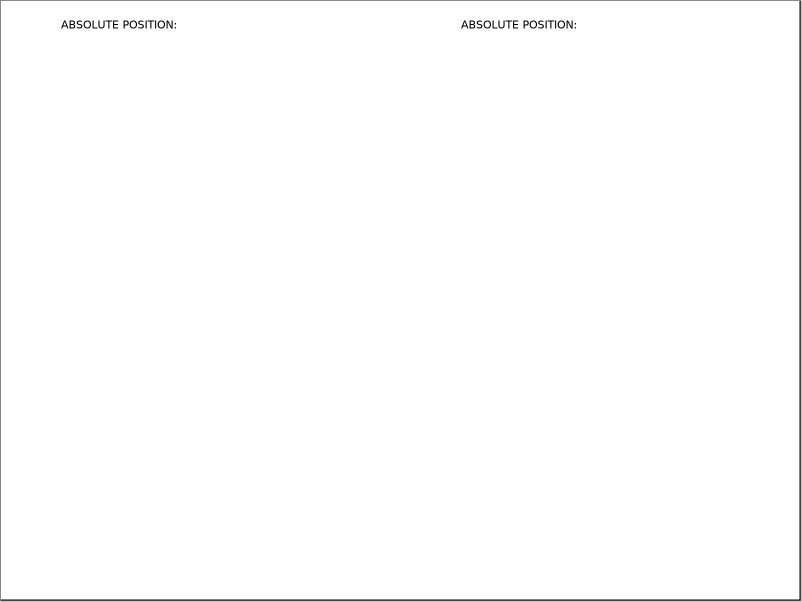
VISUALIZATION F04_Read_Axis_Error  // 802x602
    Rectangle (0,0 800x600)
    Label (10,10 170x30), "ABSOLUTE POSITION:"
    Label (410,10 170x30), "ABSOLUTE POSITION:"
END_VISUALIZATION

(* stored: Version 1.1.0.1, ProductVersion 3.1.4022.7
   Visu F04_Read_Axis_Error: Id {947bdf2a-c66b-4a9c-adb9-151978a2abad} *)
